PROGRAM PRG_EtherCAT_1_SIM
VAR
END_VAR

END_PROGRAM

(* stored: Version 1.1.0.1, ProductVersion 3.1.4026.19
   POU PRG_EtherCAT_1_SIM: Id {2deadc72-4796-4adf-b62b-ab61029111db}, SpecialFunc None *)
